DATA_BLOCK "ST10_Flow25_HShaftLoad&Unload_iDB"
{ S7_Optimized_Access := 'TRUE' }
VERSION : 0.1
NON_RETAIN
// ATTRIBUTES
// AUTO_NUMBER = False
// BLOCK_NUMBER = 1095
// END_ATTRIBUTES
"ST10_Flow25_HShaftLoad&Unload"

BEGIN

END_DATA_BLOCK

